FUNCTION_BLOCK TcoDriveSimple EXTENDS TcoCore.TcoComponent IMPLEMENTS ITcoDriveSimple
VAR_INPUT
	inEnable			:	BOOL;
	inEnablePositive	:	BOOL;
	inEnableNegative	: 	BOOL;
	inCalibrationCam	:	BOOL;
END_VAR
VAR_OUTPUT
END_VAR
VAR_IN_OUT
	inoAxisRef	: TcoAxisRef;
END_VAR


VAR
	{attribute 'hide'}
	_axisRef			:	REFERENCE TO TcoAxisRef;
	{attribute 'hide'}
	_mcReadStatus		:	Tc2_MC2.MC_ReadStatus;
	{attribute 'hide'}
	_mcPower        	:	Tc2_MC2.MC_Power;
	{attribute 'hide'}
 	_override 			:	LREAL := 100.0;
	{attribute clr [ReadOnly()]}
 	_axisStatus			:	TcoAxisStatus;
END_VAR

VAR
	_resetTask			:	ResetTask(THIS^);
	_soEResetTask		:	SoEResetTask(THIS^);
	_setPositionTask	:	SetPositionTask(THIS^);
	_homeTask			:	HomeTask(THIS^);
	_moveVelocityTask	:	MoveVelocityTask(THIS^);
	_stopTask			:	StopTask(THIS^);
	_haltTask			:	HaltTask(THIS^);
	_moveRelativeTask	:	MoveRelativeTask(THIS^);
	_moveAbsoluteTask	:	MoveAbsoluteTask(THIS^);
	_moveModuloTask		:	MoveModuloTask(THIS^);
END_VAR

IF NOT __ISVALIDREF(inoAxisRef) THEN
	Messenger.Post('Invalid reference',TcoCore.eMessageCategory.ProgrammingError);
	RETURN;
END_IF

_axisRef REF= inoAxisRef;

_mcReadStatus(Axis := _axisRef, Enable	:= TRUE);

UpdateAxisStatus();

_mcPower(	Axis			:=	_axisRef, 
			Enable			:=	inEnable, 
			Enable_Positive	:=	inEnablePositive, 
			Enable_Negative	:=	inEnableNegative, 
			Override		:=	_override, 
			BufferMode		:=	Tc2_MC2.MC_BufferMode.MC_Aborting);

_resetTask();	

_soEResetTask();

_setPositionTask();

_homeTask();

_moveVelocityTask();

_stopTask();

_haltTask();

_moveRelativeTask();

_moveAbsoluteTask();

_moveModuloTask();

PROPERTY AxisRef : REFERENCE TO TcoAxisRef
GET
IF __ISVALIDREF(_axisRef) THEN
	AxisRef REF= _axisRef;
END_IF;
END_GET
END_PROPERTY

PROPERTY AxisStatus : TcoAxisStatus
GET
UpdateAxisStatus();

AxisStatus := _axisStatus;
END_GET
END_PROPERTY

PROPERTY DriveRef : REFERENCE TO TcoDriveSimple
GET
DriveRef REF= THIS^;
END_GET
END_PROPERTY

METHOD Halt : ITcoTaskStatus
VAR_INPUT
	inDeceleration	:	LREAL;
	inJerk			:	LREAL;	
END_VAR
Halt := THIS^._haltTask.InvokeWithParams(	inDeceleration	:=	inDeceleration,
											inJerk			:=	inJerk);
END_METHOD

PROPERTY HaltTask : TcoCore.ITcoTaskStatus
GET
HaltTask := _haltTask;
END_GET
END_PROPERTY

METHOD Home : ITcoTaskStatus
VAR_INPUT
	inPosition			:	LREAL;
	inHomingMode		:	eHomingMode;
	inClearPositionLag	:	BOOL;
	inSearchDirection	:	eDirection;
	inSearchVelocity	:	LREAL;
	inSyncDirection		:	eDirection;
	inSyncVelocity		:	LREAL;
	inReferenceMode		:	eEncoderReferenceMode;
END_VAR
VAR
	_homingMode			:	Tc2_MC2.MC_HomingMode;
	_SearchDirection	:	Tc2_MC2.MC_Direction;
	_SyncDirection		:	Tc2_MC2.MC_Direction;
	_ReferenceMode		:	Tc2_MC2.E_EncoderReferenceMode;
	_message			:	STRING(125);
	
END_VAR
IF NOT Tco_TO_Tc2MC2_HomingMode(inHomingMode,_homingMode) THEN
	_message := Tc2_Standard.CONCAT('Unable to cast inHomingMode variable of type TcoDrivesBeckhoff.eHomingMode (', TO_STRING(inHomingMode));
	_message :=	Tc2_Standard.CONCAT(_message,') to the type Tc2_MC2.MC_HomingMode!!!');
	THIS^.Messenger.Post(_message,TcoCore.eMessageCategory.ProgrammingError);
	RETURN;
END_IF

IF NOT Tco_TO_Tc2MC2_Direction(inSearchDirection,_SearchDirection) THEN
	_message := Tc2_Standard.CONCAT('Unable to cast inSearchDirection variable of type TcoDrivesBeckhoff.eDirection (', TO_STRING(inSearchDirection));
	_message :=	Tc2_Standard.CONCAT(_message,') to the type Tc2_MC2.MC_Direction!!!');
	THIS^.Messenger.Post(_message,TcoCore.eMessageCategory.ProgrammingError);
	RETURN;
END_IF

IF NOT Tco_TO_Tc2MC2_Direction(inSyncDirection,_SyncDirection) THEN
	_message := Tc2_Standard.CONCAT('Unable to cast inSyncDirection variable of type TcoDrivesBeckhoff.eDirection (', TO_STRING(inSyncDirection));
	_message :=	Tc2_Standard.CONCAT(_message,') to the type Tc2_MC2.MC_Direction!!!');
	THIS^.Messenger.Post(_message,TcoCore.eMessageCategory.ProgrammingError);
	RETURN;
END_IF

IF NOT Tco_TO_Tc2MC2_EncRefMode(inReferenceMode,_ReferenceMode) THEN
	_message := Tc2_Standard.CONCAT('Unable to cast inReferenceMode variable of type TcoDrivesBeckhoff.eEncoderReferenceMode (', TO_STRING(inReferenceMode));
	_message :=	Tc2_Standard.CONCAT(_message,') to the type Tc2_MC2.E_EncoderReferenceMode!!!');
	THIS^.Messenger.Post(_message,TcoCore.eMessageCategory.ProgrammingError);
	RETURN;
END_IF

Home := THIS^._homeTask.InvokeWithParams(	inPosition			:=	inPosition,  
											inHomingMode		:=	_homingMode, 
											inClearPositionLag	:=	inClearPositionLag,
											inSearchDirection	:=	_SearchDirection,
											inSearchVelocity	:=	inSearchVelocity,
											inSyncDirection		:=	_SyncDirection,
											inSyncVelocity		:=	inSyncVelocity,
											inReferenceMode		:=	_ReferenceMode);
END_METHOD

PROPERTY HomeTask : TcoCore.ITcoTaskStatus
GET
HomeTask := _homeTask;
END_GET
END_PROPERTY

PROPERTY IsEnabled : BOOL
GET
IsEnabled := inEnable AND THIS^._mcPower.Status;
END_GET
END_PROPERTY

PROPERTY IsEnabledNegative : BOOL
GET
IsEnabledNegative := inEnableNegative;
END_GET
END_PROPERTY

PROPERTY IsEnabledPositive : BOOL
GET
IsEnabledPositive := inEnablePositive;
END_GET
END_PROPERTY

METHOD MoveAbsolute : ITcoTaskStatus
VAR_INPUT
	inPosition		:	LREAL;
	inVelocity		:	LREAL;
	inAcceleration	:	LREAL;
	inDeceleration	:	LREAL;
	inJerk			:	LREAL;	
END_VAR
MoveAbsolute := THIS^._moveAbsoluteTask.InvokeWithParams(	inPosition		:=	inPosition,
															inVelocity		:=	inVelocity,
															inAcceleration	:=	inAcceleration,
															inDeceleration	:=	inDeceleration,
															inJerk			:=	inJerk);
END_METHOD

PROPERTY MoveAbsoluteTask : TcoCore.ITcoTaskStatus
GET
MoveAbsoluteTask := _moveAbsoluteTask;
END_GET
END_PROPERTY

METHOD MoveModulo : ITcoTaskStatus
VAR_INPUT
	inPosition		:	LREAL;
	inVelocity		:	LREAL;
	inAcceleration	:	LREAL;
	inDeceleration	:	LREAL;
	inJerk			:	LREAL;	
	inDirection		:	eDirection;
END_VAR
VAR
	_direction		:	Tc2_MC2.MC_Direction;
	_message		:	STRING(125);
END_VAR
IF NOT Tco_TO_Tc2MC2_Direction(inDirection,_direction) THEN
	_message := Tc2_Standard.CONCAT('Unable to cast inDirection variable of type TcoDrivesBeckhoff.eDirection (', TO_STRING(inDirection));
	_message :=	Tc2_Standard.CONCAT(_message,') to the type Tc2_MC2.MC_Direction!!!');
	THIS^.Messenger.Post(_message,TcoCore.eMessageCategory.ProgrammingError);
	RETURN;
END_IF

MoveModulo := THIS^._moveModuloTask.InvokeWithParams(	inPosition		:=	inPosition,
														inVelocity		:=	inVelocity,
														inAcceleration	:=	inAcceleration,
														inDeceleration	:=	inDeceleration,
														inJerk			:=	inJerk,
														inDirection		:=	_direction);
END_METHOD

PROPERTY MoveModuloTask : TcoCore.ITcoTaskStatus
GET
MoveModuloTask := _moveModuloTask;
END_GET
END_PROPERTY

METHOD MoveRelative : ITcoTaskStatus
VAR_INPUT
	inDistance		:	LREAL;
	inVelocity		:	LREAL;
	inAcceleration	:	LREAL;
	inDeceleration	:	LREAL;
	inJerk			:	LREAL;	
END_VAR
MoveRelative := THIS^._moveRelativeTask.InvokeWithParams(	inDistance		:=	inDistance,
															inVelocity		:=	inVelocity,
															inAcceleration	:=	inAcceleration,
															inDeceleration	:=	inDeceleration,
															inJerk			:=	inJerk);
END_METHOD

PROPERTY MoveRelativeTask : TcoCore.ITcoTaskStatus
GET
MoveRelativeTask := _moveRelativeTask;
END_GET
END_PROPERTY

METHOD MoveVelocity : ITcoTaskStatus
VAR_INPUT
	inVelocity		:	LREAL;
	inAcceleration	:	LREAL;
	inDeceleration	:	LREAL;
	inJerk			:	LREAL;	
	inDirection		:	eDirection;
END_VAR
VAR
	_direction		:	Tc2_MC2.MC_Direction;
	_message		:	STRING(125);
END_VAR
IF NOT Tco_TO_Tc2MC2_Direction(inDirection,_direction) THEN
	_message := Tc2_Standard.CONCAT('Unable to cast inDirection variable of type TcoDrivesBeckhoff.eDirection (', TO_STRING(inDirection));
	_message :=	Tc2_Standard.CONCAT(_message,') to the type Tc2_MC2.MC_Direction!!!');
	THIS^.Messenger.Post(_message,TcoCore.eMessageCategory.ProgrammingError);
	RETURN;
END_IF

MoveVelocity := THIS^._moveVelocityTask.InvokeWithParams(	inVelocity		:=	inVelocity,
															inAcceleration	:=	inAcceleration,
															inDeceleration	:=	inDeceleration,
															inJerk			:=	inJerk,
															inDirection		:=	_direction);
END_METHOD

PROPERTY MoveVelocityTask : TcoCore.ITcoTaskStatus
GET
MoveVelocityTask := _moveVelocityTask;
END_GET
END_PROPERTY

PROPERTY Override : LREAL
GET
Override := _override;
END_GET
SET
_override := Override;
END_SET
END_PROPERTY

METHOD Reset : ITcoTaskStatus
Reset := THIS^._resetTask.Invoke();
END_METHOD

PROPERTY ResetTask : TcoCore.ITcoTaskStatus
GET
ResetTask := _resetTask;
END_GET
END_PROPERTY

(*~
	<docu>
		<summary>
			Restores this instance to the Ready state. Can be called explicitly or from within one of the restore mechanisms.	
		</summary>			
	</docu>	
~*)
METHOD  Restore : ITcoRestorable
IF __ISVALIDREF(_axisRef) THEN
	_mcPower(Axis := _axisRef, Enable := FALSE);
	_mcReadStatus(Axis:= _axisRef, Enable	:= FALSE); 
END_IF

_override := 100;

_resetTask.Restore();
_soEResetTask.Restore();
_setPositionTask .Restore();
_homeTask.Restore();
_moveVelocityTask.Restore();
_stopTask.Restore();
_haltTask.Restore();
_moveRelativeTask.Restore();
_moveAbsoluteTask.Restore();
_moveModuloTask.Restore();
END_METHOD

(*~
	<docu>
		<summary>
		    Custom service (manual, maintenance) logic.
			This method must be implemented in derived class.
		</summary>			
	</docu>	
~*)
METHOD PROTECTED  ServiceMode
END_METHOD

METHOD SetPosition : ITcoTaskStatus
VAR_INPUT
	inPosition		:	LREAL;
	inMode			:	BOOL;
END_VAR
SetPosition := THIS^._setPositionTask.InvokeWithParams(	inPosition		:=	inPosition,
														inMode			:=	inMode);
END_METHOD

PROPERTY SetPositionTask : TcoCore.ITcoTaskStatus
GET
SetPositionTask := _setPositionTask;
END_GET
END_PROPERTY

METHOD SoEReset : ITcoTaskStatus
SoEReset := THIS^._soEResetTask.Invoke();
END_METHOD

PROPERTY SoEResetTask : TcoCore.ITcoTaskStatus
GET
SoEResetTask := _soEResetTask;
END_GET
END_PROPERTY

METHOD Stop : ITcoTaskStatus
VAR_INPUT
	inDeceleration	:	LREAL;
	inJerk			:	LREAL;	
END_VAR
Stop := THIS^._stopTask.InvokeWithParams(	inDeceleration	:=	inDeceleration,
											inJerk			:=	inJerk);
END_METHOD

PROPERTY StopTask : TcoCore.ITcoTaskStatus
GET
StopTask := _stopTask;
END_GET
END_PROPERTY

METHOD INTERNAL UpdateAxisStatus
VAR
	_message : STRING(125);
END_VAR

_axisStatus.ActPos               := AxisRef.NcToPlc.ActPos;
_axisStatus.ModuloActPos         := AxisRef.NcToPlc.ModuloActPos;
_axisStatus.ModuloActTurns       := AxisRef.NcToPlc.ModuloActTurns;
_axisStatus.ActVelo              := AxisRef.NcToPlc.ActVelo;  
_axisStatus.ActAcc               := AxisRef.NcToPlc.ActAcc;  
_axisStatus.ActTorque            := AxisRef.NcToPlc.ActTorque;
_axisStatus.CmdNo                := AxisRef.NcToPlc.CmdNo;    
_axisStatus.CmdState             := AxisRef.NcToPlc.CmdState; 

IF NOT Tc2MC2_TO_Tco_AxisStates(AxisRef.Status.MotionState, _axisStatus.MotionState) THEN
	_message := Tc2_Standard.CONCAT('Unable to cast AxisRef.Status.MotionState variable of type Tc2_MC2.MC_AxisStates (', TO_STRING(AxisRef.Status.MotionState));
	_message :=	Tc2_Standard.CONCAT(_message,') to the type TcoDrivesBeckhoff.eAxisStates!!!');
	THIS^.Messenger.Post(_message,TcoCore.eMessageCategory.ProgrammingError);
END_IF

_axisStatus.Error                := AxisRef.Status.Error;                
_axisStatus.ErrorId              := AxisRef.Status.ErrorId;              
_axisStatus.ErrorStop            := AxisRef.Status.ErrorStop;            
_axisStatus.Disabled             := AxisRef.Status.Disabled;             
_axisStatus.Stopping             := AxisRef.Status.Stopping;             
_axisStatus.StandStill           := AxisRef.Status.StandStill;           
_axisStatus.DiscreteMotion       := AxisRef.Status.DiscreteMotion;       
_axisStatus.ContinuousMotion     := AxisRef.Status.ContinuousMotion;     
_axisStatus.SynchronizedMotion   := AxisRef.Status.SynchronizedMotion;   
_axisStatus.Homing               := AxisRef.Status.Homing;               
_axisStatus.ConstantVelocity     := AxisRef.Status.ConstantVelocity;     
_axisStatus.Accelerating         := AxisRef.Status.Accelerating;         
_axisStatus.Decelerating         := AxisRef.Status.Decelerating;         
_axisStatus.Operational          := AxisRef.Status.Operational;          
_axisStatus.ControlLoopClosed    := AxisRef.Status.ControlLoopClosed;    
_axisStatus.HasJob               := AxisRef.Status.HasJob;               
_axisStatus.HasBeenStopped       := AxisRef.Status.HasBeenStopped;       
_axisStatus.NewTargetPosition    := AxisRef.Status.NewTargetPosition;    
_axisStatus.InPositionArea       := AxisRef.Status.InPositionArea;       
_axisStatus.InTargetPosition     := AxisRef.Status.InTargetPosition;     
_axisStatus.Homed                := AxisRef.Status.Homed;                
_axisStatus.HomingBusy           := AxisRef.Status.HomingBusy;           
_axisStatus.MotionCommandsLocked := AxisRef.Status.MotionCommandsLocked; 
_axisStatus.SoftLimitMinExceeded := AxisRef.Status.SoftLimitMinExceeded; 
_axisStatus.SoftLimitMaxExceeded := AxisRef.Status.SoftLimitMaxExceeded; 
_axisStatus.Moving               := AxisRef.Status.Moving;               
_axisStatus.PositiveDirection    := AxisRef.Status.PositiveDirection;    
_axisStatus.NegativeDirection    := AxisRef.Status.NegativeDirection;    
_axisStatus.NotMoving            := AxisRef.Status.NotMoving;            
_axisStatus.Compensating         := AxisRef.Status.Compensating;         
_axisStatus.ExtSetPointGenEnabled:= AxisRef.Status.ExtSetPointGenEnabled;
_axisStatus.ExternalLatchValid   := AxisRef.Status.ExternalLatchValid;   
_axisStatus.CamDataQueued        := AxisRef.Status.CamDataQueued;        
_axisStatus.CamTableQueued       := AxisRef.Status.CamTableQueued;       
_axisStatus.CamScalingPending    := AxisRef.Status.CamScalingPending;    
_axisStatus.CmdBuffered          := AxisRef.Status.CmdBuffered;          
_axisStatus.PTPmode              := AxisRef.Status.PTPmode;              
_axisStatus.DriveDeviceError     := AxisRef.Status.DriveDeviceError;     
_axisStatus.IoDataInvalid        := AxisRef.Status.IoDataInvalid;        
_axisStatus.Coupled              := AxisRef.Status.Coupled;      
        
_axisStatus.OpMode.PositionAreaMonitoring   :=	AxisRef.Status.OpMode.PositionAreaMonitoring 	;
_axisStatus.OpMode.TargetPositionMonitoring :=	AxisRef.Status.OpMode.TargetPositionMonitoring  ;
_axisStatus.OpMode.LoopMode                 :=	AxisRef.Status.OpMode.LoopMode                  ;
_axisStatus.OpMode.MotionMonitoring         :=	AxisRef.Status.OpMode.MotionMonitoring          ;
_axisStatus.OpMode.PEHTimeMonitoring        :=	AxisRef.Status.OpMode.PEHTimeMonitoring         ;
_axisStatus.OpMode.BacklashCompensation     :=	AxisRef.Status.OpMode.BacklashCompensation      ;
_axisStatus.OpMode.Modulo                   :=	AxisRef.Status.OpMode.Modulo                    ;
_axisStatus.OpMode.PositionLagMonitoring    :=	AxisRef.Status.OpMode.PositionLagMonitoring     ;
_axisStatus.OpMode.VelocityLagMonitoring    :=	AxisRef.Status.OpMode.VelocityLagMonitoring     ;
_axisStatus.OpMode.SoftLimitMinMonitoring   :=	AxisRef.Status.OpMode.SoftLimitMinMonitoring    ;
_axisStatus.OpMode.SoftLimitMaxMonitoring   :=	AxisRef.Status.OpMode.SoftLimitMaxMonitoring    ;
_axisStatus.OpMode.PositionCorrection       :=	AxisRef.Status.OpMode.PositionCorrection        ;
END_METHOD

END_FUNCTION_BLOCK

(* stored: Version 1.1.0.1, ProductVersion 3.1.4024.6
   POU TcoDriveSimple: Id {e1d88b92-8a8a-0e74-0555-7cc06fb367e3}, SpecialFunc None
   Folder Axis: Id {d7605e2c-2fb5-0437-2ec5-266a0c7dda7d}
   Folder Motion: Id {9515ec36-620f-055e-2ead-75815f8c7157}
   Property AxisRef: Id {9addb9b6-186b-0d94-195f-26fedd5a4a18}
   Get Get: Id {d6e47ff9-0f85-0d36-2b20-674079d02a12}
   Property AxisStatus: Id {9f534259-f47a-013c-016f-57eedebf76e7}
   Get Get: Id {f9fdffde-5f54-0445-0964-dc68d9a08f3c}
   Property DriveRef: Id {3800d624-5130-0c3a-22c9-8c42027a5bf8}
   Get Get: Id {f663277e-3c9f-02d1-3d1a-bc1c267140dd}
   Method Halt: Id {06b4c873-3aa4-03d0-22c1-6924d11db75b}
   Property HaltTask: Id {721ccc2a-8cb6-094a-16a1-751262a37bc7}
   Get Get: Id {7f728bc9-46dc-0a19-2179-b1de30aba7b0}
   Method Home: Id {3416c275-ea54-0bdf-3bf7-9e6742cd2a7c}
   Property HomeTask: Id {3ab56154-4a39-02f0-1548-06459fed21f1}
   Get Get: Id {2bb3fbff-b440-0928-0b83-8952b6850e93}
   Property IsEnabled: Id {280b02f2-a96c-00f4-06dc-f0cc9119d0d1}
   Get Get: Id {1993ae19-9e9a-0563-1e60-73ac2e003c87}
   Property IsEnabledNegative: Id {76136ee5-e1ba-0451-0802-d036fd3e174c}
   Get Get: Id {55242dae-4611-059b-0438-765b90d6b286}
   Property IsEnabledPositive: Id {6ca8e7ee-2a04-02f9-0eb7-b131fef8ba81}
   Get Get: Id {ee313c31-0c0e-082a-0fec-4c8f300a64ca}
   Method MoveAbsolute: Id {7c866b31-0c32-0194-3f88-7187373816e9}
   Property MoveAbsoluteTask: Id {17ebba7a-d013-0a5a-3a28-1097559062ec}
   Get Get: Id {ded087e0-b1eb-0fc7-0ec1-7018b2b40a87}
   Method MoveModulo: Id {60533808-bfc3-020d-1ddf-a4a1eafb4401}
   Property MoveModuloTask: Id {86367453-a7b7-08da-0f92-37c1eae8b91a}
   Get Get: Id {9f7f478d-7d5d-06b9-3c5d-cc876e9a6f76}
   Method MoveRelative: Id {cc6ab8a3-fc1f-041a-330f-7b967a6efc54}
   Property MoveRelativeTask: Id {8caccdea-e800-07be-0faa-ea524d879ae5}
   Get Get: Id {1518a26a-d0f6-0ef4-19fc-8a061b698389}
   Method MoveVelocity: Id {1bc3a166-148c-03f6-0943-0e69683b0c9e}
   Property MoveVelocityTask: Id {540cc01c-f652-0632-29f6-354dc831965b}
   Get Get: Id {a782dff3-7d28-0c61-1597-2dc6bca94aef}
   Property Override: Id {7e6937a0-4ba3-05b0-2930-caf46da04f03}
   Get Get: Id {b2639d12-3057-054a-1e0b-10829b617131}
   Set Set: Id {2bdc560a-6a3d-00ec-3ff9-9a9b8c70e5f8}
   Method Reset: Id {b7749f10-c738-0ee2-388c-b27c2482f791}
   Property ResetTask: Id {5950371b-5e88-0c27-3e74-bb65429d19c1}
   Get Get: Id {18e492cf-625f-03ba-1857-c1a0603df608}
   Method Restore: Id {cb4df5d0-872f-0def-03a7-f8bfc3720272}
   Method ServiceMode: Id {f2dcab5e-74c4-0882-12e2-82e083006063}
   Method SetPosition: Id {e0b984cb-4674-021d-1559-4672196bcb8d}
   Property SetPositionTask: Id {e749923d-00ef-0fe7-3af7-6d91b222f204}
   Get Get: Id {db47f5b6-d402-0ac2-1e5b-5cf22a990886}
   Method SoEReset: Id {7430d658-985b-0e2d-3ddc-c2f5991b2139}
   Property SoEResetTask: Id {3d28e97c-fa27-04e2-2319-822ccba8f6af}
   Get Get: Id {e8334689-57fb-0ddc-06dd-40ce8545ba95}
   Method Stop: Id {a2b4d263-a695-059c-192f-27eca075d880}
   Property StopTask: Id {38310ba4-95f6-0e90-0216-0427029c6246}
   Get Get: Id {11ea129d-b40e-074d-138d-7e8f23c9682f}
   Method UpdateAxisStatus: Id {b151254e-094a-082e-0d80-afd3b3fd89f9} *)
